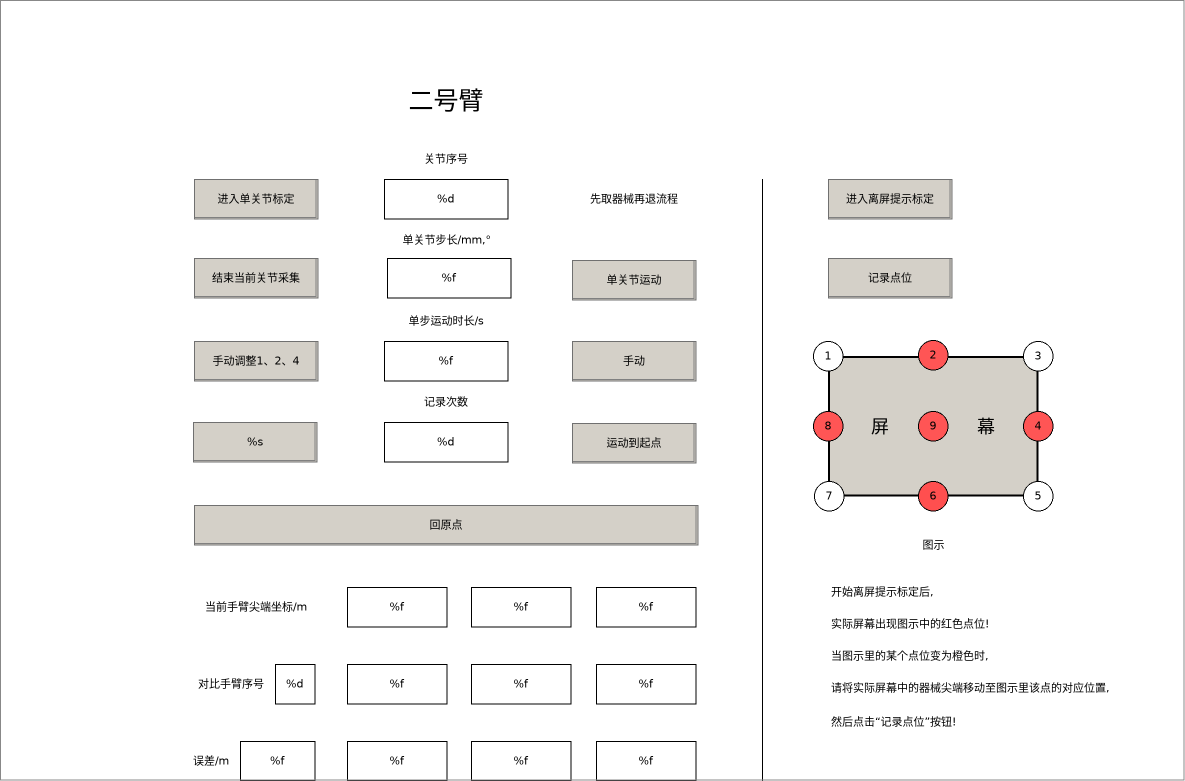
VISUALIZATION kineCali_a2  // 1185x781
    Button (194,179 124x40), "进入单关节标定", colour toggle: g_singleJntTest.m_enterSingleJntTestMode[2]
        toggle g_singleJntTest.m_enterSingleJntTestMode[2]
    Button (572,341 124x40), "手动", colour toggle: g_singleJntTest.m_manualAdjustFlag
    Button (572,423 124x40), "运动到起点", colour toggle: g_singleJntTest.m_move2StartFlag
    Rectangle (384,422 124x40), "%d", text variable: g_singleJntTest.m_dataRecordCount[2]
        OnMouseClick: write the text variable via Default, min 0, max 1000
    Label (372,220 150x40), "单关节步长/mm,°"
    Button (572,260 124x40), "单关节运动", colour toggle: g_singleJntTest.m_singleJntFlag
    Label (371,139 150x40), "关节序号"
    Rectangle (387,258 124x40), "%f", text variable: g_singleJntTest.m_jntStep
        OnMouseClick: write the text variable via Default, min 0
    Button (193,422 124x40), "%s", text variable: g_singleJntTest.m_dataRecordText, colour toggle: g_singleJntTest.m_dataRecordFlag[2]
        tap g_singleJntTest.m_dataRecordFlag[2]
    Rectangle (384,179 124x40), "%d", text variable: g_singleJntTest.m_kineCaliJntIdx
        OnMouseClick: write the text variable via Default, min 1, max 8
    Button (194,505 504x40), "回原点", colour toggle: g_singleJntTest.m_return2OriginFlag
        toggle g_singleJntTest.m_return2OriginFlag
    Rectangle (384,341 124x40), "%f", text variable: g_singleJntTest.m_EndT
        OnMouseClick: write the text variable via Default, min 0, max 100
    Label (371,301 150x40), "单步运动时长/s"
    Label (371,382 150x40), "记录次数"
    Label (384,79 124x43), "二号臂"
    Button (194,258 124x40), "结束当前关节采集", colour toggle: g_singleJntTest.m_manualEndFlag
        toggle g_singleJntTest.m_manualEndFlag
    Button (194,341 124x40), "手动调整1、2、4", colour toggle: g_singleJntTest.m_manual124StartFlag
        toggle g_singleJntTest.m_manual124StartFlag
    Label (572,179 124x40), "先取器械再退流程"
    Rectangle (347,587 100x40), "%f", text variable: g_singleJntTest.m_instruPose[2].m_pos[1]
        OnMouseClick: write the text variable via Default, min 0, max 100
    Rectangle (471,587 100x40), "%f", text variable: g_singleJntTest.m_instruPose[2].m_pos[2]
        OnMouseClick: write the text variable via Default, min 0, max 100
    Rectangle (596,587 100x40), "%f", text variable: g_singleJntTest.m_instruPose[2].m_pos[3]
        OnMouseClick: write the text variable via Default, min 0, max 100
    Rectangle (347,664 100x40), "%f", text variable: g_singleJntTest.m_instruPoseAnother.m_pos[1]
        OnMouseClick: write the text variable via Default, min 0, max 100
    Rectangle (471,664 100x40), "%f", text variable: g_singleJntTest.m_instruPoseAnother.m_pos[2]
        OnMouseClick: write the text variable via Default, min 0, max 100
    Rectangle (596,664 100x40), "%f", text variable: g_singleJntTest.m_instruPoseAnother.m_pos[2]
        OnMouseClick: write the text variable via Default, min 0, max 100
    Rectangle (275,664 40x40), "%d", text variable: g_singleJntTest.m_instruAnotherIdx
        OnMouseClick: write the text variable via Default, min 0, max 4
    Label (191,664 80x40), "对比手臂序号"
    Label (191,587 130x40), "当前手臂尖端坐标/m"
    Rectangle (347,741 100x40), "%f", text variable: g_singleJntTest.m_instruPoseError[2].m_pos[1]
        OnMouseClick: write the text variable via Default, min 0, max 100
    Rectangle (471,741 100x40), "%f", text variable: g_singleJntTest.m_instruPoseError[2].m_pos[2]
        OnMouseClick: write the text variable via Default, min 0, max 100
    Rectangle (596,741 100x40), "%f", text variable: g_singleJntTest.m_instruPoseError[2].m_pos[3]
        OnMouseClick: write the text variable via Default, min 0, max 100
    Rectangle (240,741 75x40), "%f", text variable: g_singleJntTest.m_instruErrDis[2]
        OnMouseClick: write the text variable via Default, min 0, max 4
    Label (191,741 40x40), "误差/m"
    Button (828,179 124x40), "进入离屏提示标定", colour toggle: g_offScreenTest.m_enterSingleJntTestMode[2]
        toggle g_singleJntTest.m_enterSingleJntTestMode[1]
    Line (762,179) (762,781)
    Button (828,258 124x40), "记录点位", text variable: g_singleJntTest.m_dataRecordText, colour toggle: g_offScreenTest.m_dataRecordFlag[2]
        tap g_offScreenTest.m_dataRecordFlag[2]
    Rectangle (828,356 210x140), colour variable: m_offScreenTest.m_caliPointEndFlag[1]
    Ellipse (813,341 30x30), "1", colour variable: m_offScreenTest.m_caliPointEndFlag[1]
        p2167032090: m_offScreenTest.m_caliPointStartFlag[1]
    Label (865,412 30x30), "屏"
    Label (971,412 30x30), "幕"
    Ellipse (918,340 30x30), "2", colour variable: m_offScreenTest.m_caliPointEndFlag[2]
        p2167032090: m_offScreenTest.m_caliPointStartFlag[2]
    Ellipse (1023,411 30x30), "4", colour variable: m_offScreenTest.m_caliPointEndFlag[4]
        p2167032090: m_offScreenTest.m_caliPointStartFlag[4]
    Ellipse (1023,481 30x30), "5", colour variable: m_offScreenTest.m_caliPointEndFlag[5]
        p2167032090: m_offScreenTest.m_caliPointStartFlag[5]
    Ellipse (918,481 30x30), "6", colour variable: m_offScreenTest.m_caliPointEndFlag[6]
        p2167032090: m_offScreenTest.m_caliPointStartFlag[6]
    Ellipse (814,481 30x30), "7", colour variable: m_offScreenTest.m_caliPointEndFlag[7]
        p2167032090: m_offScreenTest.m_caliPointStartFlag[7]
    Ellipse (813,411 30x30), "8", colour variable: m_offScreenTest.m_caliPointEndFlag[8]
        p2167032090: m_offScreenTest.m_caliPointStartFlag[8]
    Ellipse (918,411 30x30), "9", colour variable: m_offScreenTest.m_caliPointEndFlag[1]
        p2167032090: m_offScreenTest.m_caliPointStartFlag[1]
    Ellipse (1023,341 30x30), "3", colour variable: m_offScreenTest.m_caliPointEndFlag[3]
        p2167032090: m_offScreenTest.m_caliPointStartFlag[3]
    Label (828,646 216x20), "当图示里的某个点位变为橙色时,"
    Label (828,678 357x20), "请将实际屏幕中的器械尖端移动至图示里该点的对应位置,"
    Label (828,614 216x20), "实际屏幕出现图示中的红色点位!"
    Label (828,582 216x20), "开始离屏提示标定后,"
    Label (828,712 216x20), "然后点击“记录点位”按钮!"
    Label (918,535 31x20), "图示"
END_VISUALIZATION

(* stored: Version 1.1.0.1, ProductVersion 3.1.4024.11
   Visu kineCali_a2: Id {91accdc4-27ce-4135-afbd-5b06ea0dbc33} *)
